TYPE ST_Point3D :
STRUCT
    X : LREAL;
    Y : LREAL;
    Z : LREAL;
END_STRUCT
END_TYPE

(* stored: Version 1.1.0.1, ProductVersion 3.1.4026.20
   DUT ST_Point3D: Id {4ee37b51-d703-4e7e-911c-1e3623d3bb67} *)
